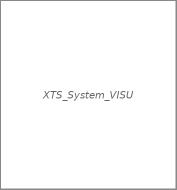
VISUALIZATION Visualization  // 177x190
    Frame (0,0 177x190)
        shows XTS_System_VISU(xts := MAIN.fbXTSSystem)
END_VISUALIZATION

(* stored: Version 1.1.0.1, ProductVersion 3.1.4024.11
   Visu Visualization: Id {527ffa00-3a93-4fd0-aad7-a32ea8a3eae2} *)
